(* CODESYS project xLH_base_io_ethercat_FINAL_00_10.project
   Description: Receives some incoming messages and echoes them with CAN-ID +1
   Title: CAN Bus API Example
   Version: 1.0.0.0
   Company: 3S - Smart Software Solutions GmbH
   Author: 3S - Smart Software Solutions GmbH

Project tree, tasks and I/O mapping:
  XLH_base : CODESYS Control for Raspberry Pi 64 SL, CODESYS, order no. 2302000009, version 4.12.0.0
    application app
      libraries: Standard, 3.5.18.0 (System); Memory, * (3S - Smart Software Solutions GmbH); Util, 3.5.19.0 (System); VisuDialogs, * (System); CAA Tick Extern, 3.5.17.0 (CAA Technical Workgroup); SysTime, 3.5.17.0 (System); CmpIecTask, * (System); xemax Bibliothek, 0.20 (xemax ag)
      task MAIN_TASK (cyclic, interval 20 ms, priority 0) calls MAIN, io, IO_ETHERCAT
      task EtherCAT_Task (cyclic, interval t#4ms, priority 1) calls nothing
      program io [ST]
      program MAIN [ST]
      program IO_ETHERCAT [FBD]
    SoftMotion General Axis Pool
    GPIOs_A_B : GPIOs B+/Pi2, CODESYS, version 4.12.0.0
        input  app.io.bSw1 : BOOL  // digital inputs (GPIO0..GPIO31).Bit4
        input  app.io.bSw2 : BOOL  // digital inputs (GPIO0..GPIO31).Bit5
        input  app.io.bSw3 : BOOL  // digital inputs (GPIO0..GPIO31).Bit6
        input  app.io.bSw4 : BOOL  // digital inputs (GPIO0..GPIO31).Bit12
        input  app.io.bSw5 : BOOL  // digital inputs (GPIO0..GPIO31).Bit13
        input  app.io.bSw6 : BOOL  // digital inputs (GPIO0..GPIO31).Bit16
        input  app.io.bSw7 : BOOL  // digital inputs (GPIO0..GPIO31).Bit17
        input  app.io.bSw8 : BOOL  // digital inputs (GPIO0..GPIO31).Bit19
        output app.io.bLed1 : BOOL  // digital outputs (GPIO0..GPIO31).Bit20
        output app.io.bLed2 : BOOL  // digital outputs (GPIO0..GPIO31).Bit21
        output app.io.bLed3 : BOOL  // digital outputs (GPIO0..GPIO31).Bit22
        output app.io.bLed4 : BOOL  // digital outputs (GPIO0..GPIO31).Bit23
        output app.io.bLed5 : BOOL  // digital outputs (GPIO0..GPIO31).Bit24
        output app.io.bLed6 : BOOL  // digital outputs (GPIO0..GPIO31).Bit26
        output app.io.bLed7 : BOOL  // digital outputs (GPIO0..GPIO31).Bit27
        unmapped channels: digital inputs (GPIO0..GPIO31), digital outputs (GPIO0..GPIO31)
    Onewire
    Camera device
      <Leer>
    SPI
    I²C
    EtherCAT_Master : EtherCAT Master, CODESYS, version 4.7.0.0
        settings: NetworkName = 'eth0'; NetworkName = "eth0"; SrcAddress1 = 224; SrcAddress2 = 1278612855
      EK1100 : EK1100 EtherCAT-Koppler (2A E-Bus), Beckhoff Automation GmbH & Co. KG, order no. EK1100, version Revision=16#00120000
          settings: DC sync0 cycletime = 4000; DC sync1 cycletime = 4000
        EL1004 : EL1004 4K. Dig. Eingang 24V, 3ms, Beckhoff Automation GmbH & Co. KG, order no. EL1004, version Revision=16#00130000
            settings: DC sync0 cycletime = 4000; DC sync1 cycletime = 4000
            input  app.IO_ETHERCAT.bEl1004_1_0 : BIT  // Input
            unmapped channels: Input, Input, Input
        EL1004_1 : EL1004 4K. Dig. Eingang 24V, 3ms, Beckhoff Automation GmbH & Co. KG, order no. EL1004, version Revision=16#00130000
            settings: DC sync0 cycletime = 4000; DC sync1 cycletime = 4000
            unmapped channels: Input, Input, Input, Input
        EL2004 : EL2004 4K. Dig. Ausgang 24V, 0.5A, Beckhoff Automation GmbH & Co. KG, order no. EL2004, version Revision=16#00120000
            settings: DC sync0 cycletime = 4000; DC sync1 cycletime = 4000
            output app.IO_ETHERCAT.bEL2004_1_0 : BIT  // Output
            unmapped channels: Output, Output, Output
        EL2004_1 : EL2004 4K. Dig. Ausgang 24V, 0.5A, Beckhoff Automation GmbH & Co. KG, order no. EL2004, version Revision=16#00120000
            settings: DC sync0 cycletime = 4000; DC sync1 cycletime = 4000
            unmapped channels: Output, Output, Output, Output
        EL3162 : EL3162 2K. Ana. Eingang 0-10V, Beckhoff Automation GmbH & Co. KG, order no. EL3162, version Revision=16#00130000
            unmapped channels: Status, Value, Status, Value
        EL4004 : EL4004 4K. Ana. Ausgang 0-10V, 12bit, Beckhoff Automation GmbH & Co. KG, order no. EL4004, version Revision=16#00150000
            unmapped channels: Analog output, Analog output, Analog output, Analog output
  libraries: VisuSymbols, 4.5.0.0 (System); DepictorBase, 1.0.5.0 (3S - Smart Software Solutions GmbH)
  text list GlobalTextList
*)

// XLH_base/app/MAIN
PROGRAM MAIN
VAR
	vVersionPlc: VERSION;
	sVersionPlc: STRING(255);
	vVersionLib: VERSION;
	sVersionLib: STRING(255);
END_VAR

// Version Bibliothex xemax
vVersionPlc.uiMajor := 1;
vVersionPlc.uiMinor := 0;
sVersionPlc := CONCAT(TO_STRING(TO_UINT(vVersionPlc.uiMajor)), CONCAT('.', (TO_STRING(TO_UINT(vVersionPlc.uiMinor)))));
vVersionLib := xemax.GetLibVersion();
sVersionLib := CONCAT(TO_STRING(TO_UINT(vVersionLib.uiMajor)), CONCAT('.', (TO_STRING(TO_UINT(vVersionLib.uiMinor)))));

(*
==================================================================================================
Login Codesys in die xLH - SPS 
user: xlh
pw: xlh
==================================================================================================
*)

END_PROGRAM

// XLH_base/app/io
PROGRAM io
VAR_INPUT			
	bLed1: BOOL;
	bLed2: BOOL;
	bLed3: BOOL;
	bLed4: BOOL;
	bLed5: BOOL;
	bLed6: BOOL;
	bLed7: BOOL;	
	oled: OLED;
END_VAR
VAR_OUTPUT
	bSw1: BOOL;
	bSw2: BOOL;
	bSw3: BOOL;
	bSw4: BOOL;
	bSw5: BOOL;
	bSw6: BOOL;
	bSw7: BOOL;
	bSw8: BOOL;
END_VAR
VAR
END_VAR

xemax.LOCAL_TIME_AND_TIME_ZONE();
xemax.TASK_INFO();
oled();

END_PROGRAM

// XLH_base/app/IO_ETHERCAT
PROGRAM IO_ETHERCAT
VAR_INPUT
	bEl1004_1_0: BOOL;
END_VAR
VAR_OUTPUT
	bEL2004_1_0: BOOL;
END_VAR
VAR
	fbBlink: BLINK;
	bDummy: BOOL;
END_VAR

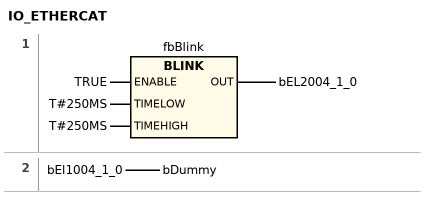
// NETWORK 1
fbBlink(ENABLE := TRUE, TIMELOW := T#250MS, TIMEHIGH := T#250MS); // BLINK
bEL2004_1_0 := fbBlink.OUT;

// NETWORK 2
bDummy := bEl1004_1_0;

END_PROGRAM
